Staubli VAL3: KILLTASK.pgx

public program KillTask()
begin



  if taskStatus("Move")!=-1
    taskKill("Move")
  endIf
  if taskStatus("ReadFile")!=-1
    taskKill("ReadFile")
  endIf

  if taskStatus("Preset")!=-1
    taskKill("Preset")
  endIf

  if taskStatus("WeldEnd")!=-1
    taskKill("WeldEnd")
  endIf

end
